// TIA Portal V17 export
// export: Created 2026-04-13T11:12:45.3578854Z, ExportSetting WithDefaults, DisplayName Totally Integrated Automation Portal, DisplayVersion V17 Update 4, DisplayName TIA Portal Openness, DisplayVersion V17 Update 4, DisplayName TIA Portal Version Control Interface, DisplayVersion V17, DisplayName SINAMICS Startdrive Advanced, DisplayVersion V17, DisplayName SINAMICS Startdrive G130, G150, S120, S150, SINAMICS MV, S210, DisplayVersion V17, DisplayName SINAMICS Startdrive G110M, G120, G120C, G120D, G120P, G115D, DisplayVersion V17, DisplayName STEP 7 Professional, DisplayVersion V17 Update 4, DisplayName STEP 7 Safety, DisplayVersion V17, DisplayName WinCC Professional, DisplayVersion V17 Update 4
VAR_GLOBAL   // PLC tag table "IOM"
   QSF送风机 AT %M300.0 : Bool;
   QSF送风机风扇 AT %M300.1 : Bool;
   QDJ电加热器 AT %M301.1 : Bool;
   QSS输送风机 AT %M301.2 : Bool;
   QSS输送加热器 AT %M301.3 : Bool;
   QYF引风机 AT %M300.2 : Bool;
   QYF引风机风扇 AT %M300.3 : Bool;
   QLX离心雾化 AT %M300.4 : Bool;
   QLX离心雾化风扇 AT %M300.5 : Bool;
   QLX离心雾化油泵 AT %M300.6 : Bool;
   QJL进料泵 AT %M300.7 : Bool;
   QJL进料泵风扇 AT %M301.0 : Bool;
   QFM蜂鸣器 AT %M301.4 : Bool;
   QZS指示灯 AT %M301.5 : Bool;
   QYS钥匙开关 AT %M301.6 : Bool;
   QZM照明灯 AT %M301.7 : Bool;
   QPH平衡比例调节阀 AT %M302.0 : Bool;
   QCC除尘脉冲 AT %M302.1 : Bool;
   QJF进风蒸汽比例调节阀 AT %M302.2 : Bool;
   QHF回风蒸汽调节阀 AT %M302.3 : Bool;
   QBY备用1 AT %M302.4 : Bool;
   QBY备用2 AT %M302.5 : Bool;
   QBY备用3 AT %M302.6 : Bool;
   QBY备用4 AT %M302.7 : Bool;
   QXY泄压阀 AT %M303.0 : Bool;
   QJF进风冷却水阀 AT %M303.1 : Bool;
   QSS输送进风阀 AT %M303.2 : Bool;
   QQL气流雾化阀 AT %M303.3 : Bool;
   QKS开式排风隔断阀 AT %M303.4 : Bool;
   QBS闭式排风隔断阀 AT %M303.5 : Bool;
   QKS开式进风隔断阀 AT %M303.6 : Bool;
   QBS闭式进风隔断阀 AT %M303.7 : Bool;
   QYJ一级冷却水阀 AT %M304.0 : Bool;
   QEJ二级冷冻水阀 AT %M304.1 : Bool;
   QYJ一级排液阀 AT %M304.2 : Bool;
   QEJ二级排液阀 AT %M304.3 : Bool;
   QCW除雾排液阀 AT %M304.4 : Bool;
   QRJ溶剂回收排放阀 AT %M304.5 : Bool;
   QZT主塔气锤1 AT %M304.6 : Bool;
   QZT主塔气锤2 AT %M304.7 : Bool;
   QZT主塔气锤3 AT %M305.0 : Bool;
   QZT主塔气锤4 AT %M305.1 : Bool;
   QASA室内回水阀 AT %M305.2 : Bool;
   QYJ一级缓存振荡器 AT %M305.3 : Bool;
   QASA室外回水阀 AT %M305.4 : Bool;
   QEJ二级缓存震荡器 AT %M305.5 : Bool;
   QCC除尘气锤1 AT %M305.6 : Bool;
   QCC除尘气锤2 AT %M305.7 : Bool;
   QCC除尘缓存震荡器 AT %M306.0 : Bool;
   QRJ溶剂排液泵进阀 AT %M306.1 : Bool;
   QSN室内清洗总阀 AT %M306.2 : Bool;
   QBD补氮阀 AT %M306.3 : Bool;
   QJD进氮阀 AT %M306.4 : Bool;
   QJF进风蒸汽开关阀 AT %M306.5 : Bool;
   QJF进风蒸汽排水阀 AT %M306.6 : Bool;
   QLG料罐清洗阀 AT %M306.7 : Bool;
   QQX清洗溶剂出阀 AT %M307.0 : Bool;
   QWL物料进阀 AT %M307.1 : Bool;
   QYJ一级出料上阀 AT %M307.2 : Bool;
   QYJ一级出料下阀 AT %M307.3 : Bool;
   QEJ二级出料上阀 AT %M307.4 : Bool;
   QEJ二级出料下阀 AT %M307.5 : Bool;
   QCC除尘出料上阀 AT %M307.6 : Bool;
   QCC除尘出料下阀 AT %M307.7 : Bool;
   QHF回风蒸汽开关阀 AT %M308.0 : Bool;
   QHF回风蒸汽排水阀 AT %M308.1 : Bool;
   QSS输送出料上阀 AT %M308.2 : Bool;
   QSS输送出料下阀 AT %M308.3 : Bool;
   QTD塔顶清洗球阀 AT %M308.4 : Bool;
   QQG气缸升降阀 AT %M308.5 : Bool;
   QZT主塔清洗进水阀 AT %M308.6 : Bool;
   QXF旋风管道清洗阀 AT %M308.7 : Bool;
   QYJ一级旋风清洗阀 AT %M309.0 : Bool;
   QEJ二级旋风清洗阀 AT %M309.1 : Bool;
   QCC除尘管道清洗阀 AT %M309.2 : Bool;
   QCC除尘清洗阀 AT %M309.3 : Bool;
   QSS输送管路清洗阀 AT %M309.4 : Bool;
   QLC料仓清洗阀 AT %M309.5 : Bool;
   QJR加热清洗阀 AT %M309.6 : Bool;
   QWK蜗壳清洗阀 AT %M309.7 : Bool;
   QCF出风高效清洗阀 AT %M310.0 : Bool;
   QZT主塔排水阀 AT %M310.1 : Bool;
   QSS输送管路排水阀 AT %M310.2 : Bool;
   QLC料仓清洗排水阀 AT %M310.3 : Bool;
   QSF送风机清洗阀 AT %M310.4 : Bool;
   QYF引风机清洗阀 AT %M310.5 : Bool;
   QYJ一级冷凝清洗阀 AT %M310.6 : Bool;
   QEJ二级冷凝清洗阀 AT %M310.7 : Bool;
   QSF送风机排水阀 AT %M311.0 : Bool;
   QYF引风机排水阀 AT %M311.1 : Bool;
   ISF送风机 AT %M350.0 : Bool;
   IYF引风机 AT %M350.1 : Bool;
   ILX离心雾化器 AT %M350.2 : Bool;
   IJL进料泵 AT %M350.3 : Bool;
   IDJ电加热 AT %M350.4 : Bool;
   ISF输送风机 AT %M350.5 : Bool;
   ISF输送加热 AT %M350.6 : Bool;
   IJT急停 AT %M350.7 : Bool;
   ILQ冷却水流量 AT %M351.0 : Bool;
   ILD冷冻水流量 AT %M351.1 : Bool;
   IJF进风冷却水流量 AT %M351.2 : Bool;
   IPY排液流量 AT %M351.3 : Bool;
   IBD补氮阀开反馈 AT %M351.4 : Bool;
   IBD补氮阀关反馈 AT %M351.5 : Bool;
   IJD进氮阀开反馈 AT %M351.6 : Bool;
   IJD进氮阀关反馈 AT %M351.7 : Bool;
   IXY泄压阀开反馈 AT %M352.0 : Bool;
   IXY泄压阀关反馈 AT %M352.1 : Bool;
   IQL气流雾化阀开反馈 AT %M352.2 : Bool;
   IQL气流雾化阀关反馈 AT %M352.3 : Bool;
   ISF输送进风阀开反馈 AT %M352.4 : Bool;
   ISF输送进风阀关反馈 AT %M352.5 : Bool;
   IKS开式排风隔断阀开反馈 AT %M352.6 : Bool;
   IKS开式排风隔断阀关反馈 AT %M352.7 : Bool;
   IBS闭式排风隔断阀开反馈 AT %M353.0 : Bool;
   IBS闭式排风隔断阀关反馈 AT %M353.1 : Bool;
   IKS开式进风隔断阀开反馈 AT %M353.2 : Bool;
   IKS开式进风隔断阀关反馈 AT %M353.3 : Bool;
   IBS闭式进风隔断阀开反馈 AT %M353.4 : Bool;
   IBS闭式进风隔断阀关反馈 AT %M353.5 : Bool;
   IYJ一级冷却水阀开反馈 AT %M353.6 : Bool;
   IYJ一级冷却水阀关反馈 AT %M353.7 : Bool;
   IEJ二级冷冻水阀开反馈 AT %M354.0 : Bool;
   IEJ二级冷冻水阀关反馈 AT %M354.1 : Bool;
   IYJ一级排液阀开反馈 AT %M354.2 : Bool;
   IYJ一级排液阀关反馈 AT %M354.3 : Bool;
   IEJ二级排液阀开反馈 AT %M354.4 : Bool;
   IEJ二级排液阀关反馈 AT %M354.5 : Bool;
   ICW除雾排液阀开反馈 AT %M354.6 : Bool;
   ICW除雾排液阀关反馈 AT %M354.7 : Bool;
   IRJ溶剂回收排放阀开反馈 AT %M355.0 : Bool;
   IRJ溶剂回收排放阀关反馈 AT %M355.1 : Bool;
   IJF进风冷却水阀开反馈 AT %M355.2 : Bool;
   IJF进风冷却水阀关反馈 AT %M355.3 : Bool;
   ITD塔顶清洗球阀开反馈 AT %M355.4 : Bool;
   ITD塔顶清洗球阀关反馈 AT %M355.5 : Bool;
   IQX清洗伸缩气缸降反馈 AT %M355.6 : Bool;
   IQX清洗伸缩气缸升反馈 AT %M355.7 : Bool;
   QRS热水洗请求 AT %M311.2 : Bool;
   QRJ溶剂洗 AT %M311.3 : Bool;
   QBY备用7 AT %M311.4 : Bool;
   QSN室内排水隔膜泵 AT %M311.5 : Bool;
   QRJ溶剂排液泵 AT %M311.6 : Bool;
   QBY备用10 AT %M311.7 : Bool;
   QBY备用11 AT %M312.0 : Bool;
   QBY备用12 AT %M312.1 : Bool;
   QBY备用13 AT %M312.2 : Bool;
   QBY备用14 AT %M312.3 : Bool;
   QBY备用15 AT %M312.4 : Bool;
   QBY备用16 AT %M312.5 : Bool;
   QBY备用17 AT %M312.6 : Bool;
   QBY备用18 AT %M312.7 : Bool;
   QBY备用19 AT %M313.0 : Bool;
   QBY备用20 AT %M313.1 : Bool;
   QQG气缸升 AT %M313.2 : Bool;
   QQG气缸降 AT %M313.3 : Bool;
   QBD布袋振打1 AT %M313.4 : Bool;
   QSB设备振打 AT %M313.5 : Bool;
   QBD布袋振打3 AT %M313.6 : Bool;
   QBD布袋振打4 AT %M313.7 : Bool;
   QYH氧含仪隔断阀 AT %M314.0 : Bool;
   QHS回水隔断阀1 AT %M314.1 : Bool;
   IJF进风保护温度 AT %M356.0 : Bool;
   ISS输送保护温度 AT %M356.1 : Bool;
   IBP爆破片1反馈 AT %M356.2 : Bool;
   IBP爆破片2反馈 AT %M356.3 : Bool;
   ISN室内排水开反馈 AT %M356.4 : Bool;
   ISN室内排水关反馈 AT %M356.5 : Bool;
   IRJ溶剂排液泵开反馈 AT %M356.6 : Bool;
   IRJ溶剂排液泵关反馈 AT %M356.7 : Bool;
   QXT心跳发送信号 AT %M314.2 : Bool;
   QCS纯水洗请求 AT %M314.3 : Bool;
   QJS碱水洗请求 AT %M314.4 : Bool;
   QRJ溶剂请求 AT %M314.5 : Bool;
   QYG压干请求 AT %M314.6 : Bool;
   QQZ前置水阀 AT %M314.7 : Bool;
   QYJ一级旋风振打锤 AT %M315.0 : Bool;
   QEJ二级旋风振打锤 AT %M315.1 : Bool;
   QYJ一级旋风振荡器 AT %M315.2 : Bool;
   QCIP启动 AT %M315.3 : Bool;
   QGS供水泵启动 AT %M315.4 : Bool;
   QZS注射水洗 AT %M315.5 : Bool;
   QSJ水进程泵 AT %M315.6 : Bool;
   QRJ溶剂进程泵 AT %M315.7 : Bool;
   QQS缺水状态 AT %M316.0 : Bool;
   QRC热纯自动洗 AT %M316.1 : Bool;
END_VAR
